// TIA Portal V20 export
DATA_BLOCK "DB_Alarmas"   // DB3
{ S7_Optimized_Access := 'TRUE' }
// stored: MemoryReserve 100
   VAR
      Registro_Fallos : Word;
   END_VAR
BEGIN
END_DATA_BLOCK
